// TwinCAT 3 PLC project AlternateCoolingSystem
// ProgramVersion: 3.1.4024.0
// libraries:
//   Tc2_Standard, * (Beckhoff Automation GmbH)
//   Tc2_System, * (Beckhoff Automation GmbH)
//   Tc3_Module, * (Beckhoff Automation GmbH)
// project tree:
//   DUTs/ ST_Tank.TcDUT
//   / PlcTask.TcTTO
//   POUs/ FB_PressureTankController.TcPOU, FB_TankController.TcPOU, F_CheckAlarm.TcPOU (not stored), F_CoolTank.TcPOU (not stored), I_TankController.TcIO, MAIN.TcPOU
// (motion and I/O tree: see PLC project instructions_practice)
// real-time tasks:
//   TASK PlcTask: cycle T#10ms, priority 20, ADS port 350
//   TASK PlcTask1: cycle T#10ms, priority 22, ADS port 351

CONFIGURATION AlternateCoolingSystem
    RESOURCE PLC ON TwinCAT3
        TASK PlcTask(INTERVAL := T#10ms, PRIORITY := 22);
        PROGRAM MAIN WITH PlcTask : MAIN;
    END_RESOURCE
END_CONFIGURATION

// ---- DUTs/ST_Tank.TcDUT
TYPE ST_Tank :
STRUCT
	nId : INT;
	fTemperature : REAL;
	fLevel : REAL;
	bAlarm : BOOL;
END_STRUCT
END_TYPE

// ---- POUs/I_TankController.TcIO
INTERFACE I_TankController

METHOD ApplyCooling : BOOL
VAR_INPUT
END_VAR
END_METHOD

METHOD CheckSafety : BOOL
VAR_INPUT
END_VAR
END_METHOD

METHOD StartController
VAR_INPUT
END_VAR
END_METHOD

END_INTERFACE

// ---- POUs/MAIN.TcPOU
PROGRAM MAIN
VAR
	stTank1 : ST_Tank := (nId := 101,fTemperature := 80.3, fLevel := 80, bAlarm := FALSE );
	stTank2 : ST_Tank  := (nId := 102,fTemperature := 72.5, fLevel := 70, bAlarm := FALSE );
	stTank3 : ST_Tank  := (nId := 103,fTemperature := 90.8, fLevel := 90, bAlarm := FALSE );
	
	fbController1 : FB_TankController(stTank1);
	fbController2 : FB_TankController(stTank2);
	fbController3 : FB_PressureTankController(stTank3);
	
	aTankArray : ARRAY[1..cNUMBER_OF_TANKS] OF I_TankController := [fbController1, fbController2, fbController3];
	i : INT ;
	bStart : bool;
END_VAR
VAR CONSTANT
	cNUMBER_OF_TANKS :INT :=3;
END_VAR

IF bStart THEN
	FOR i := 1 TO cNUMBER_OF_TANKS DO
		IF aTankArray[i] <> 0 THEN
			aTankArray[i].StartController();
		END_IF
	END_FOR
	bStart := FALSE;
END_IF

END_PROGRAM

// ---- POUs/FB_TankController.TcPOU
FUNCTION_BLOCK FB_TankController IMPLEMENTS I_TankController

VAR
	stTank :REFERENCE TO ST_Tank;
END_VAR

{warning 'add method implementation '}
METHOD ApplyCooling : BOOL
IF stTank.bAlarm THEN
	F_CoolTank(stTank);
END_IF
END_METHOD

{warning 'add method implementation '}
METHOD CheckSafety : BOOL
IF F_CheckAlarm( pTank := ADR(stTank) ) THEN
	stTank.bAlarm := TRUE;
END_IF
END_METHOD

METHOD FB_init : BOOL
VAR_INPUT
	bInitRetains : BOOL; // if TRUE, the retain variables are initialized (warm start / cold start)
	bInCopyCode : BOOL;  // if TRUE, the instance afterwards gets moved into the copy code (online change)
	_stTank : REFERENCE TO ST_TANK;
END_VAR
stTank REF= _stTank;
END_METHOD

METHOD StartController
VAR_INPUT
END_VAR
IF __ISVALIDREF(stTank) THEN
	CheckSafety();
	ApplyCooling();

	IF NOT stTank.bAlarm THEN
		stTank.fTemperature := stTank.fTemperature + 5;
	END_IF
END_IF
END_METHOD

END_FUNCTION_BLOCK

// ---- POUs/FB_PressureTankController.TcPOU
FUNCTION_BLOCK FB_PressureTankController EXTENDS FB_TankController
VAR_INPUT
END_VAR
VAR_OUTPUT
END_VAR
VAR
END_VAR

METHOD ControlPressure 
VAR_INPUT
END_VAR
END_METHOD

METHOD StartController
VAR_INPUT
END_VAR
SUPER^.StartController();
ControlPressure();
END_METHOD

END_FUNCTION_BLOCK
